// TIA Portal V18 export
// export: Created 2025-12-01T17:51:11.6599994Z, ExportSetting None, DisplayName Totally Integrated Automation Portal, DisplayVersion V18 Update 5, DisplayName TIA Portal Openness, DisplayVersion V18 Update 5, DisplayName TIA Portal Teamcenter Gateway, DisplayVersion V18, DisplayName TIA Portal Version Control Interface, DisplayVersion V18, DisplayName STEP 7 Professional, DisplayVersion V18 Update 5, DisplayName STEP 7 Safety, DisplayVersion V18, DisplayName WinCC Professional, DisplayVersion V18 Update 5
DATA_BLOCK "IAI_A1"   // DB2211
{ S7_Optimized_Access := 'FALSE' }
// stored: AutoNumber false
   VAR RETAIN
      In : Struct
         iInterlock : Bool;   // interlock
         "iManJog+" : Bool;   // positive motion/action/...manually
         "iManJog-" : Bool;   // negtive motion/action/...manually
         iAutoStart : Bool;   // negtive motion/action/...automaticly
         iHome : Bool;   // Homing
         iCancelTask : Bool;   // Cancel task
         iPauseTask : Bool;   // Pause task
         iManStart : Bool;   // positive motion/action/...automaticly
         iManListStart : Bool;
         iLimitSwitchActive : Bool := true;
         iLimitSoftActive : Bool := true;
         iRunningTimeout : Time;
         iHomingTimeout : Time;
         iAutoPosition : DInt;
         iAutoVelocity : Int;
         iManListPosition : DInt;
         iManListVelocity : Int;
         iManListNumber : Int;   // position list number
         iManPosition : DInt;
         iManVelocity : Int;
         iMode : Int;   // 1-相对;2-绝对
      END_STRUCT;
      Out : Struct
         oReady : Bool;
         oWarning : Bool;   // warning
         oError : Bool;   // error
         oInterlock : Bool;
         oServoEnable : Bool;
         oRunning : Bool;
         oHoming : Bool;
         oHomeRef : Bool;
         oServoPosOK : Bool;
         oErrorCode : Int;
         oStatus : Int;
         oActPosition : DInt;
         oManualListPos : DInt;
      END_STRUCT;
      IO : Struct
         ioManEnale : Bool;
         ioAutoEnale : Bool;
      END_STRUCT;
      Spare : Struct
         S : Array[0..100] of Byte;
      END_STRUCT;
      Manual : Struct
         Index : Int := 1;
         Pos : Array[1..20] of Struct
            Pos : Real;
            Vel : Int;
         END_STRUCT;
      END_STRUCT;
      Auto : Struct
         Index : Int := 1;
         Pos : Array[1..20] of Struct
            Pos : Real;
            Vel : Int;
         END_STRUCT;
      END_STRUCT;
      Interlock : Struct
         Active : Bool;
         Case1 : Bool;
         Case2 : Bool;
         Case3 : Bool;
         Case4 : Bool;
         Case5 : Bool;
         Case6 : Bool;
         Case7 : Bool;
         Case8 : Bool;
         Case9 : Bool;
         Case10 : Bool;
      END_STRUCT;
      PositionOk : Array[1..20] of Bool;
      Home_Pos : Struct
         "Home Pos Pls" : Bool;
         "Arrow indication" : Int;
         "Process prompt" : Int;
         "Button prompt" : Int;
      END_STRUCT;
   END_VAR
BEGIN
   // Auto.Pos[1] : 1.取料位置
   // Auto.Pos[2] : 2.放料位置
   // Auto.Pos[3] : 3.
   // Auto.Pos[4] : 4.
   // Auto.Pos[5] : 5.
   // Auto.Pos[6] : 6.
   // Auto.Pos[7] : 7.
   // Auto.Pos[8] : 8.
   // Auto.Pos[9] : 9.
   // PositionOk[1] : [1]
   // PositionOk[2] : [2]
   // PositionOk[3] : [3]
   // PositionOk[4] : [4]
   // PositionOk[5] : [5]
   // PositionOk[6] : [6]
   // PositionOk[7] : [7]
   // PositionOk[8] : [8]
   // PositionOk[9] : [9]
END_DATA_BLOCK
